(*

## Short summary

This interface provides assert statements for strings
For UTF-16 strings up to 255 ``WORD`` (``WSTRING(Tc2_System.MAX_STRING_LENGTH)``) use the property `IStringAssertions.utf16`.
For windows-125x strings up to 255 ``BYTE`` (``Tc2_System.T_MaxString``) use the property `IStringAssertions.windows125x`.
For windows-125x or UTF-16 strings that are longer, use the property `IStringAssertions.anyString`  

.. <legal notes>

legal notes
=================
| SPDX-FileCopyrightText: © 2022 ekvip automation GmbH <info@ekvip.de>
| SPDX-License-Identifier: Apache-2.0
| For details check: Apache-2.0_

.. _Apache-2.0: https://www.apache.org/licenses/LICENSE-2.0

.. </legal notes>

properties
==================

*)

INTERFACE IStringAssertions EXTENDS __SYSTEM.IQueryInterface

(*

## Short summary
Returns an interface `IUnicodeStringAssertions` with assert statements,
for UTF-8 and UTF-16 strings with an undefined length.

**Attention:** 
	All strings are handled as null terminated byte/word streams.
	For UTF-8 is end of the string 16#00
	For UTF-16 is end of the string 16#00_00

**Attention:** 
	The interface `IUnicodeAssertions` uses ``ANY_STRING``, 
	for this it's not possible to use literals/constants,
	because for ``ANY`` types generates the compiler ``__SYSTEM.AnyType``
	and ``__SYSTEM.AnyType`` contains a pointer  

.. <legal notes>

legal notes
=================
| SPDX-FileCopyrightText: © 2022 ekvip automation GmbH <info@ekvip.de>
| SPDX-License-Identifier: Apache-2.0
| For details check: Apache-2.0_

.. _Apache-2.0: https://www.apache.org/licenses/LICENSE-2.0

.. </legal notes>

*)

PROPERTY unicode :IUnicodeStringAssertions
GET
END_GET
END_PROPERTY

(*

## Short summary
Returns an interface `IUtf16StringAssertions` with assert statements
for UTF-16 strings up to 255 ``WORD`` length (``WSTRING(Tc2_System.MAX_STRING_LENGTH)``)

.. <legal notes>

legal notes
=================
| SPDX-FileCopyrightText: © 2022 ekvip automation GmbH <info@ekvip.de>
| SPDX-License-Identifier: Apache-2.0
| For details check: Apache-2.0_

.. _Apache-2.0: https://www.apache.org/licenses/LICENSE-2.0

.. </legal notes>

*)

PROPERTY utf16 :IUtf16StringAssertions
GET
END_GET
END_PROPERTY

(*

## Short summary
Returns an interface `IUtf8StringAssertions` with assert statements
for UTF-8 strings up to 255 bytes length (``STRING(Tc2_System.MAX_STRING_LENGTH)``)

.. <legal notes>

legal notes
=================
| SPDX-FileCopyrightText: © 2022 ekvip automation GmbH <info@ekvip.de>
| SPDX-License-Identifier: Apache-2.0
| For details check: Apache-2.0_

.. _Apache-2.0: https://www.apache.org/licenses/LICENSE-2.0

.. </legal notes>

*)

PROPERTY utf8 :IUtf8StringAssertions
GET
END_GET
END_PROPERTY

(*

## Short summary
Returns an interface `IWindows125xStringAssertions` with assert statements for 8-bit 
windows-1252 and windows-1251 strings up to 255 characters length (``Tc2_System.T_MaxString``).
Use Tc2_Utilities.GLOBAL_SBCS_TABLE variable to select required encoding

.. <legal notes>

legal notes
=================
| SPDX-FileCopyrightText: © 2022 ekvip automation GmbH <info@ekvip.de>
| SPDX-License-Identifier: Apache-2.0
| For details check: Apache-2.0_

.. _Apache-2.0: https://www.apache.org/licenses/LICENSE-2.0

.. </legal notes>

*)

PROPERTY windows125x :IWindows125xStringAssertions
GET
END_GET
END_PROPERTY

END_INTERFACE

(* stored: Version 1.1.0.1, ProductVersion 3.1.4026.11
   Itf IStringAssertions: Id {e18995ab-9503-4af3-9fad-9e2f0d75cae0}
   Property unicode: Id {a6d1bf92-b879-42a6-b334-cbeb0b424f47}
   Get Get: Id {4858134d-4f7a-4114-ba99-44e92d0dc761}
   Property utf16: Id {8df4010b-3eae-4a2e-8150-ce528203d304}
   Get Get: Id {56969a66-6e5c-4612-8909-a36d80986004}
   Property utf8: Id {2345ac52-5459-4b86-a402-9aada8a6f95d}
   Get Get: Id {02366ac8-9231-4e2e-9f14-9970d0a7d8f7}
   Property windows125x: Id {4575868b-605a-448b-bf27-f4ae1935dcfb}
   Get Get: Id {083c4bed-972f-42b1-9291-b49d3e49c543} *)
